// TIA Portal V18 export
VAR_GLOBAL   // PLC tag table "AI"
   "H/SSR_019_TT01_IN" AT %IW70 : Int;
   "H/SSR_019_TT02_IN" AT %IW72 : Int;
   "H/SSR_019_APT01_IN" AT %IW74 : Int;
   "H/SSR_019_GPT101_IN" AT %IW78 : Int;
   "H/SSR_019_GPT201_IN" AT %IW80 : Int;
   "H/SSR_019_GPT301_IN" AT %IW82 : Int;
   "H/SSR_019_GPT401_IN" AT %IW84 : Int;
   "H/SSR_019_GPT501_IN" AT %IW86 : Int;
   "H/SSR_019_GPT601_IN" AT %IW88 : Int;
   "H/SSR_019_TT03_IN" AT %IW76 : Int;
   Tag_1 AT %T5 : Timer;
END_VAR
